// TIA Portal V16 export
// export: Created 2025-08-01T13:37:59.6794473Z, ExportSetting WithDefaults, DisplayName Totally Integrated Automation Portal, DisplayVersion V16, DisplayName TIA Portal Version Control Interface, DisplayVersion V16, DisplayName TIA Portal Openness, DisplayVersion V16, DisplayName STEP 7 Professional, DisplayVersion V16, DisplayName STEP 7 Safety, DisplayVersion V16, DisplayName WinCC Advanced, DisplayVersion V16
FUNCTION_BLOCK "ResetOuputs_Function"   // FB9, LAD
TITLE = Reset Ouput Functions With Commands
VERSION : 0.1
// stored: AutoNumber true, IsIECCheckEnabled false, UDAEnableTagReadback false
   VAR_INPUT
      StopCommand_NC : Bool;
      StopCommand_NO : Bool;
   END_VAR
   VAR_OUTPUT
      Output_1 : Bool;
      Output_2 : Bool;
      Output_3 : Bool;
      Output_4 : Bool;
      Output_5 : Bool;
      Output_6 : Bool;
      Output_7 : Bool;
      Output_8 : Bool;
      Output_9 : Bool;
      Output_10 : Bool;
   END_VAR
BEGIN

REGION Network 1: NW1
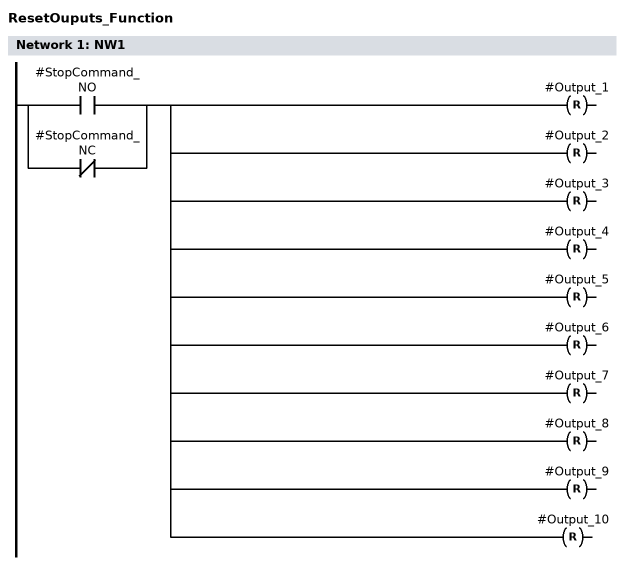
   RUNG wire#powerrail
      Contact( #StopCommand_NO )
      wire#w1
      R_Coil( #Output_1 )
   END_RUNG
   RUNG wire#powerrail
      I_Contact( #StopCommand_NC )
   END_RUNG wire#w1
   RUNG wire#w1
      R_Coil( #Output_2 )
   END_RUNG
   RUNG wire#w1
      R_Coil( #Output_3 )
   END_RUNG
   RUNG wire#w1
      R_Coil( #Output_4 )
   END_RUNG
   RUNG wire#w1
      R_Coil( #Output_5 )
   END_RUNG
   RUNG wire#w1
      R_Coil( #Output_6 )
   END_RUNG
   RUNG wire#w1
      R_Coil( #Output_7 )
   END_RUNG
   RUNG wire#w1
      R_Coil( #Output_8 )
   END_RUNG
   RUNG wire#w1
      R_Coil( #Output_9 )
   END_RUNG
   RUNG wire#w1
      R_Coil( #Output_10 )
   END_RUNG
   // the same network as SCL:
   IF #StopCommand_NO OR NOT #StopCommand_NC THEN
       #Output_1 := FALSE;
       #Output_2 := FALSE;
       #Output_3 := FALSE;
       #Output_4 := FALSE;
       #Output_5 := FALSE;
       #Output_6 := FALSE;
       #Output_7 := FALSE;
       #Output_8 := FALSE;
       #Output_9 := FALSE;
       #Output_10 := FALSE;
   END_IF;
END_REGION
END_FUNCTION_BLOCK
